{attribute addProperty BoxType "EL3403-0000-0017"}
{attribute addProperty Id "IndexAT %Q*USINT81"}
{attribute addProperty CRC "2702217147"}
{attribute addProperty SizeInBites "8"}
{attribute addProperty SizeInBytes "1"}
TYPE PM_Outputs_Channel_A1108FBB :
STRUCT
	{attribute addProperty Name "Index"}
	Index AT %Q* : USINT;
END_STRUCT
END_TYPE

(* stored: Version 1.2.0.0, ProductVersion 3.1.4024.9
   DUT PM_Outputs_Channel_A1108FBB: Id {54fd3482-915f-4104-b773-73fe23604467} *)
